// TIA Portal project "Orale_Carrello" (V15.1)

(* hardware
DEVICE "S7-1200 station_1"  S7-1200 Station
   slot 0: "Telaio di montaggio_0"  S7-1200 Rack  Rack  V1.0
   slot 1: "PLC_1"  CPU 1214C DC/DC/DC  6ES7 214-1AG40-0XB0  V4.2
*)

// ===== PLC "PLC_1"  CPU 1214C DC/DC/DC =====

VAR_GLOBAL   // PLC tag table "Tabella delle variabili standard"
   "Mup" AT %Q0.0 : Bool;
   "Mdown" AT %Q0.1 : Bool;
   "MD" AT %Q0.2 : Bool;
   "MS" AT %Q0.3 : Bool;
   "L0" AT %I0.4 : Bool;
   "L1" AT %I0.5 : Bool;
   "V1" AT %I0.6 : Bool;
   "V2" AT %I0.7 : Bool;
   "start" AT %I1.0 : Bool;
END_VAR

DATA_BLOCK "variabili_stato"   // DB1
{ S7_Optimized_Access := 'TRUE' }
VERSION : 0.1
   VAR RETAIN
      home : Bool := true;
   END_VAR
   VAR
      p1 : Bool;
      p2 : Bool;
      p0 : Bool;
      p1ritorno : Bool;
   END_VAR
BEGIN
END_DATA_BLOCK

// folder: System blocks/Program resources

DATA_BLOCK "IEC_Timer_0_DB"   // DB2
{ S7_Optimized_Access := 'TRUE' }
AUTHOR : Simatic
FAMILY : IEC
NAME : IEC_TMR
VERSION : 1.0
// stored: InstanceOfName IEC_TIMER
"IEC_TIMER"
BEGIN
END_DATA_BLOCK

// folder: (top level)

ORGANIZATION_BLOCK "Main"   // OB1, LAD, ProgramCycle
TITLE = "Main Program Sweep (Cycle)"
{ S7_Optimized_Access := 'TRUE' }
VERSION : 0.1
   VAR_INPUT
      Initial_Call : Bool;   // Initial call of this OB
      Remanence : Bool;   // =True, if remanent data are available
   END_VAR
BEGIN

REGION Network 1
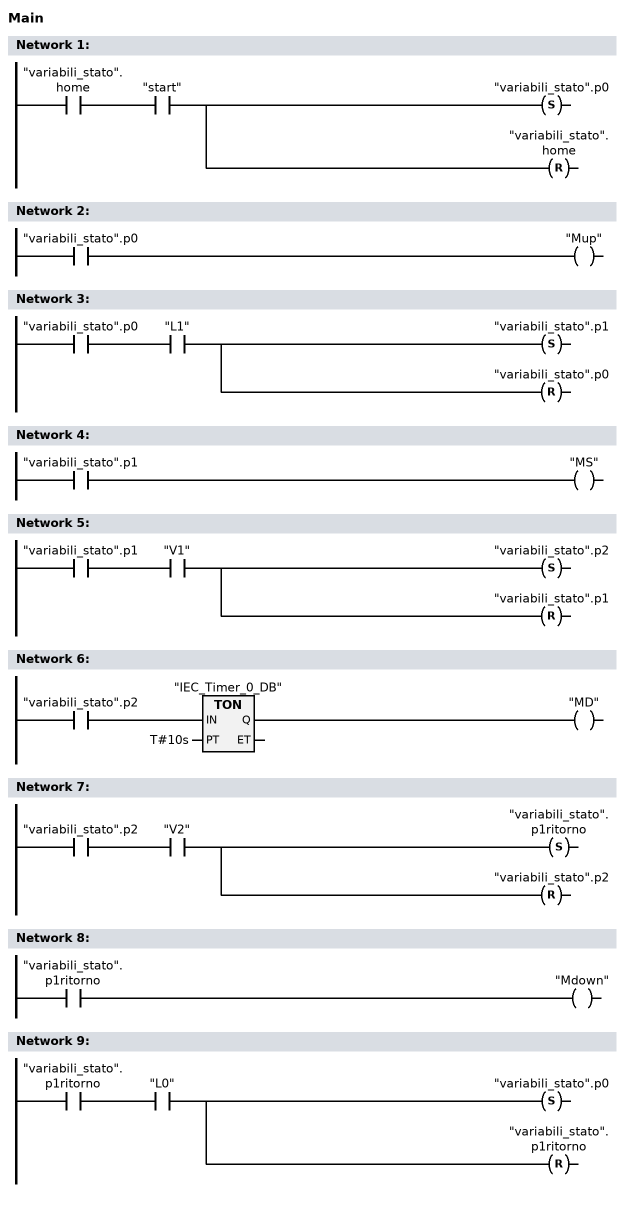
   RUNG wire#powerrail
      Contact( "variabili_stato".home )
      Contact( "start" )
      wire#w1
      S_Coil( "variabili_stato".p0 )
   END_RUNG
   RUNG wire#w1
      R_Coil( "variabili_stato".home )
   END_RUNG
   // the same network as SCL:
   IF "variabili_stato".home AND "start" THEN
       "variabili_stato".p0 := TRUE;
       "variabili_stato".home := FALSE;
   END_IF;
END_REGION

REGION Network 2
   RUNG wire#powerrail
      Contact( "variabili_stato".p0 )
      Coil( "Mup" )
   END_RUNG
   // the same network as SCL:
   "Mup" := "variabili_stato".p0;
END_REGION

REGION Network 3
   RUNG wire#powerrail
      Contact( "variabili_stato".p0 )
      Contact( "L1" )
      wire#w1
      S_Coil( "variabili_stato".p1 )
   END_RUNG
   RUNG wire#w1
      R_Coil( "variabili_stato".p0 )
   END_RUNG
   // the same network as SCL:
   IF "variabili_stato".p0 AND "L1" THEN
       "variabili_stato".p1 := TRUE;
       "variabili_stato".p0 := FALSE;
   END_IF;
END_REGION

REGION Network 4
   RUNG wire#powerrail
      Contact( "variabili_stato".p1 )
      Coil( "MS" )
   END_RUNG
   // the same network as SCL:
   "MS" := "variabili_stato".p1;
END_REGION

REGION Network 5
   RUNG wire#powerrail
      Contact( "variabili_stato".p1 )
      Contact( "V1" )
      wire#w1
      S_Coil( "variabili_stato".p2 )
   END_RUNG
   RUNG wire#w1
      R_Coil( "variabili_stato".p1 )
   END_RUNG
   // the same network as SCL:
   IF "variabili_stato".p1 AND "V1" THEN
       "variabili_stato".p2 := TRUE;
       "variabili_stato".p1 := FALSE;
   END_IF;
END_REGION

REGION Network 6
   "IEC_Timer_0_DB".TON(IN := "variabili_stato".p2, PT := T#10s);
   "MD" := "IEC_Timer_0_DB".Q;
END_REGION

REGION Network 7
   RUNG wire#powerrail
      Contact( "variabili_stato".p2 )
      Contact( "V2" )
      wire#w1
      S_Coil( "variabili_stato".p1ritorno )
   END_RUNG
   RUNG wire#w1
      R_Coil( "variabili_stato".p2 )
   END_RUNG
   // the same network as SCL:
   IF "variabili_stato".p2 AND "V2" THEN
       "variabili_stato".p1ritorno := TRUE;
       "variabili_stato".p2 := FALSE;
   END_IF;
END_REGION

REGION Network 8
   RUNG wire#powerrail
      Contact( "variabili_stato".p1ritorno )
      Coil( "Mdown" )
   END_RUNG
   // the same network as SCL:
   "Mdown" := "variabili_stato".p1ritorno;
END_REGION

REGION Network 9
   RUNG wire#powerrail
      Contact( "variabili_stato".p1ritorno )
      Contact( "L0" )
      wire#w1
      S_Coil( "variabili_stato".p0 )
   END_RUNG
   RUNG wire#w1
      R_Coil( "variabili_stato".p1ritorno )
   END_RUNG
   // the same network as SCL:
   IF "variabili_stato".p1ritorno AND "L0" THEN
       "variabili_stato".p0 := TRUE;
       "variabili_stato".p1ritorno := FALSE;
   END_IF;
END_REGION
END_ORGANIZATION_BLOCK